// TwinCAT 3 PLC project Untitled1
// Title: EventBufferLibrary
// Company: Runtimevic SL
// Author: Víctor Durán Muñoz
// ProjectVersion: 1.0.0
// Description: victorduranm@hotmail.com
// ProgramVersion: 3.1.4023.0
// libraries:
//   Tc2_Standard, * (Beckhoff Automation GmbH)
//   Tc2_System, * (Beckhoff Automation GmbH)
//   Tc2_Utilities, * (Beckhoff Automation GmbH)
//   Tc3_EventLogger, * (Beckhoff Automation GmbH)
//   Tc3_Module, * (Beckhoff Automation GmbH)
//   TcUnit, * (www.tcunit.org)
// project tree:
//   / Demostration_1.TcTTO, PlcTask.TcTTO
//   DUTs/ E_EventType.TcDUT, ST_Event.TcDUT
//   POUs/ Demostration.TcPOU, EventLogger.TcPOU, FB_CsvPersistentEventStorage.TcPOU, FB_EventBuffer.TcPOU, FB_XmlPersistentEventStorage.TcPOU, I_PersistentEventStorage.TcIO, UpdateEventTimestampWithSystemTime.TcPOU
//   Project Information/ F_GetCompany.TcPOU, F_GetTitle.TcPOU, F_GetVersion.TcPOU
//   Test/ FB_EventBuffer_Test.TcPOU, PRG_TEST.TcPOU
//   Version/ Global_Version.TcGVL
// real-time tasks:
//   TASK PlcTask: cycle T#10ms, priority 20, ADS port 350
//   TASK Demostration: cycle T#10ms, priority 2, ADS port 352

CONFIGURATION Untitled1
    RESOURCE PLC ON TwinCAT3
        TASK Demostration_1(INTERVAL := T#10ms, PRIORITY := 2);
        TASK PlcTask(INTERVAL := T#10ms, PRIORITY := 20);
        PROGRAM Demostration WITH Demostration_1 : Demostration;
        PROGRAM PRG_TEST WITH PlcTask : PRG_TEST;
    END_RESOURCE
END_CONFIGURATION

// ---- DUTs/E_EventType.TcDUT
{attribute 'qualified_only'}
{attribute 'strict'}
TYPE E_EventType :
(
	Alarm :=0,
	Message :=1
);
END_TYPE

// ---- DUTs/ST_Event.TcDUT
TYPE ST_Event :
STRUCT
	eEventType :E_EventType;
	eEventSeverity: Tc3_EventLogger.TcEventSeverity;
	nEventIdentity: UDINT;
	sEventText: STRING(255);
	dtTimestamp: DATE_AND_TIME;
END_STRUCT
END_TYPE

// ---- Version/Global_Version.TcGVL
{attribute 'TcGenerated'}
{attribute 'no-analysis'}
{attribute 'linkalways'}
// This function has been automatically generated from the project information.
VAR_GLOBAL CONSTANT
	{attribute 'const_non_replaced'}
	stLibVersion_EventBufferLibrary : ST_LibVersion := (iMajor := 1, iMinor := 0, iBuild := 0, iRevision := 0, nFlags := 0, sVersion := '1.0.0');
END_VAR

// ---- POUs/I_PersistentEventStorage.TcIO
INTERFACE I_PersistentEventStorage

METHOD StoreEvent
VAR_INPUT
	stEvent : ST_Event;
END_VAR
END_METHOD

END_INTERFACE

// ---- POUs/Demostration.TcPOU
PROGRAM Demostration
VAR
	bBoolean : BOOL := FALSE;
	
	// Event #1
	eEventType1 :E_EventType := E_EventType.Alarm;
	eEventSeverity1: Tc3_EventLogger.TcEventSeverity := Tc3_EventLogger.TcEventSeverity.Error;
	nEventIdentity1: UDINT := 42;
	sEventText1: STRING(255) := 'this is a scary event #1';
	
	// Event #2
	eEventType2 :E_EventType := E_EventType.Alarm;
	eEventSeverity2: Tc3_EventLogger.TcEventSeverity := Tc3_EventLogger.TcEventSeverity.Error;
	nEventIdentity2: UDINT := 43;
	sEventText2: STRING(255) := 'this is a scary event #2';
	
	// Event #3
	eEventType3 :E_EventType := E_EventType.Alarm;
	eEventSeverity3: Tc3_EventLogger.TcEventSeverity := Tc3_EventLogger.TcEventSeverity.Error;
	nEventIdentity3: UDINT := 44;
	sEventText3: STRING(255) := 'this is a scary event #3';	
	
	
	BufferArray : ARRAY[0..(nMAXIMUM_NUMBER_OF_EVENTS * (SIZEOF(ST_Event) + nMEMORY_RING_BUFFER_INTERNAL_EXTRA_SPACING))] OF BYTE;
	fbEventBuffer : FB_EventBuffer(ADR(BufferArray),SIZEOF(BufferArray));	
	fbXmlPersistentEventStorage : FB_XmlPersistentEventStorage;	
	fbCsvPersistentEventStorage : FB_CsvPersistentEventStorage(fbEventBuffer);
//	EventLogger : EventLogger(fbXmlPersistentEventStorage);
	EventLogger : EventLogger(fbCsvPersistentEventStorage);
END_VAR
VAR CONSTANT
	nMAXIMUM_NUMBER_OF_EVENTS : UDINT := 10; 
	nMEMORY_RING_BUFFER_INTERNAL_EXTRA_SPACING : UDINT := 8;
END_VAR

IF bBoolean THEN
	EventLogger.AddEvent(eEventType1, eEventSeverity1, nEventIdentity1, sEventText1);
	EventLogger.AddEvent(eEventType2, eEventSeverity2, nEventIdentity2, sEventText2);
	EventLogger.AddEvent(eEventType3, eEventSeverity3, nEventIdentity3, sEventText3);
//	EventLogger.AddEvent(eEventType1, eEventSeverity1, nEventIdentity1, sEventText1);
	bBoolean := FALSE;
END_IF

fbCsvPersistentEventStorage();

END_PROGRAM

// ---- POUs/FB_EventBuffer.TcPOU
FUNCTION_BLOCK FB_EventBuffer
VAR
	fbMemRingBuffer			: Tc2_Utilities.FB_MemRingBuffer;
	pPointerToArrayBuffer 	: POINTER TO BYTE;
	nSizeOfArrayBuffer    	: UDINT;
END_VAR

METHOD PUBLIC AddEvent
VAR_INPUT
	stEvent : ST_Event;
END_VAR
VAR_OUTPUT
	bOk: BOOL; //
END_VAR
fbMemRingBuffer.A_AddTail(pWrite  := ADR(stEvent),
    					  cbWrite := SIZEOF(stEvent),  					
    					  pBuffer := pPointerToArrayBuffer,
    					  cbBuffer:= nSizeOfArrayBuffer);
						  
bOk:= fbMemRingBuffer.bOk;
END_METHOD

METHOD FB_init : BOOL
VAR_INPUT
	bInitRetains : BOOL; // if TRUE, the retain variables are initialized (warm start / cold start)
	bInCopyCode : BOOL;  // if TRUE, the instance afterwards gets moved into the copy code (online change)
	pPointerToArrayBuffer : POINTER TO BYTE;
	nSizeOfArrayBuffer    : UDINT;
END_VAR
THIS^.pPointerToArrayBuffer	:= pPointerToArrayBuffer;
THIS^.nSizeOfArrayBuffer    := nSizeOfArrayBuffer;
END_METHOD

METHOD PUBLIC GetAndRemoveEvent
VAR_OUTPUT
	stEvent : ST_Event;
	bOk  : BOOL;
END_VAR
fbMemRingBuffer.A_RemoveHead (pRead  := ADR(stEvent),
    					      cbRead := SIZEOF(stEvent),  					
    					      pBuffer := pPointerToArrayBuffer,
    					      cbBuffer:= nSizeOfArrayBuffer);
						  
bOk:= fbMemRingBuffer.bOk;
END_METHOD

METHOD PUBLIC GetNumberOfEvents : UDINT
GetNumberOfEvents := fbMemRingBuffer.nCount;
END_METHOD

END_FUNCTION_BLOCK

// ---- POUs/FB_XmlPersistentEventStorage.TcPOU
FUNCTION_BLOCK FB_XmlPersistentEventStorage IMPLEMENTS I_PersistentEventStorage
VAR_INPUT
END_VAR
VAR_OUTPUT
END_VAR
VAR
END_VAR

{warning 'add method implementation '}
METHOD StoreEvent
VAR_INPUT
	stEvent	: ST_Event;
END_VAR
// Here is there XML-Writing is supposed to be done
//Were is where the FB_XmlPersistentEventStorage se debe implementar el codigo aqui.
END_METHOD

END_FUNCTION_BLOCK

// ---- POUs/FB_CsvPersistentEventStorage.TcPOU
FUNCTION_BLOCK FB_CsvPersistentEventStorage IMPLEMENTS I_PersistentEventStorage
VAR
	fbFileOpen : FB_FileOpen := (sPathName := 'C:\Events.log', 
								 nMode := FOPEN_MODEAPPEND OR FOPEN_MODETEXT);
	fbFilePuts : FB_FilePuts;	
	fbFileClose : FB_FileClose;						 
	eWriteState : (WAIT_FOR_EVENT, FILE_OPEN_TRIGGER, FILE_OPEN, WRITE_EVENT_TRIGGER, WRITE_EVENT, FILE_CLOSE_TRIGGER, FILE_CLOSE, CLEAR_FILE_FB, ERROR);
	//stEventWrittenToFile : ST_Event;
	
	CsvString : T_MaxString;
	stEventFromBuffer : ST_Event;
	fbEventBuffer : REFERENCE TO FB_EventBuffer;
	bOkIgnore : BOOL;
END_VAR

CASE eWriteState OF
	WAIT_FOR_EVENT :
		//Do Anything
		IF fbEventBuffer.GetNumberOfEvents() > 0 THEN
			eWriteState := FILE_OPEN_TRIGGER;
		END_IF
		
	FILE_OPEN_TRIGGER :
		fbFileOpen(bExecute := TRUE);
		eWriteState := FILE_OPEN;
		
	FILE_OPEN :
		IF fbFileOpen.bError THEN
			eWriteState := ERROR;
		ELSIF NOT fbFileOpen.bBusy AND fbFileOpen.hFile <> 0 THEN
			eWriteState := WRITE_EVENT_TRIGGER;
		END_IF		
            fbFileOpen(bExecute := FALSE);	
		
	WRITE_EVENT_TRIGGER :
		eWriteState := FILE_OPEN_TRIGGER;
		fbEventBuffer.GetAndRemoveEvent(stEvent=> stEventFromBuffer, bOk=>bOkIgnore);
		CsvString := CreateCsvString(stEvent := stEventFromBuffer);
		fbFilePuts(bExecute := TRUE, 
				   sLine := CsvString,
				   hFile := fbFileOpen.hFile);
		eWriteState := WRITE_EVENT;
		
	WRITE_EVENT :
		IF fbFilePuts.bError THEN
			eWriteState := ERROR;
		ELSIF NOT fbFilePuts.bBusy THEN
			eWriteState := FILE_CLOSE_TRIGGER;
		END_IF			
		fbFilePuts(bExecute := FALSE);


	FILE_CLOSE_TRIGGER :
		fbFileClose(bExecute := TRUE,
					hFile := fbFileOpen.hFile);
		eWriteState := FILE_CLOSE;
		
	FILE_CLOSE :
	    IF fbFileClose.bError THEN
		    eWriteState := ERROR;
	    ELSIF NOT fbFileClose.bBusy THEN
		    eWriteState := WAIT_FOR_EVENT;
	    END_IF
	    fbFileClose(bExecute := FALSE);

	CLEAR_FILE_FB:
		fbFileOpen(bExecute := FALSE);
		fbFilePuts(bExecute := FALSE);
		fbFileClose(bExecute := FALSE);
		eWriteState := FILE_OPEN_TRIGGER;
		
	ERROR :
		//Do Nothing
END_CASE

METHOD PRIVATE CreateCsvString : T_MaxString
VAR_INPUT
	stEvent : REFERENCE TO ST_Event;
END_VAR
VAR
	TempString : T_MaxString;
//	count:  INT;
END_VAR
//TempString := TO_STRING(count +1);
//TempString := CONCAT(STR1:= TempString, STR2:= ',');
//TempString := CONCAT(STR1:= TempString, STR2:= TO_STRING(stEvent.eEventType));

TempString := TO_STRING(stEvent.eEventType);
TempString := CONCAT(STR1:= TempString, STR2:= ',');
TempString := CONCAT(STR1:= TempString, STR2:= TO_STRING(stEvent.eEventSeverity));
TempString := CONCAT(STR1:= TempString, STR2:= ',');
TempString := CONCAT(STR1:= TempString, STR2:= TO_STRING(stEvent.nEventIdentity));
TempString := CONCAT(STR1:= TempString, STR2:= ',');
TempString := CONCAT(STR1:= TempString, STR2:=  stevent.sEventText);
TempString := CONCAT(STR1:= TempString, STR2:= ',');
TempString := CONCAT(STR1:= TempString, STR2:=  TO_STRING(stEvent.dtTimestamp));
TempString := CONCAT(STR1:= TempString, STR2:=  '$N');

CreateCsvString := TempString;
END_METHOD

METHOD FB_init : BOOL
VAR_INPUT
	bInitRetains : BOOL; // if TRUE, the retain variables are initialized (warm start / cold start)
	bInCopyCode : BOOL;  // if TRUE, the instance afterwards gets moved into the copy code (online change)
	fbEventBuffer : REFERENCE TO FB_EventBuffer;
END_VAR
THIS^.fbEventBuffer REF= fbEventBuffer;
END_METHOD


METHOD StoreEvent
VAR_INPUT
	stEvent	: ST_Event;
END_VAR
VAR
	bOkIgnore : BOOL;
END_VAR
(*
IF eWriteState = WAIT_FOR_EVENT THEN
	eWriteState := FILE_OPEN_TRIGGER;
	stEventWrittenToFile := stEvent;
END_IF
*)
fbEventBuffer.AddEvent(stEvent:= stEvent, bOk=>bOkIgnore);
END_METHOD

END_FUNCTION_BLOCK

// ---- POUs/EventLogger.TcPOU
FUNCTION_BLOCK EventLogger
VAR
	EventBuffer : ARRAY[1..MAXIMUM_SIZE_OF_EVENT_BUFFER] OF ST_Event;
	CurrentEventBufferIndex : INT :=0;
	
	_PersistentEventStorage : I_PersistentEventStorage;
END_VAR
VAR CONSTANT
	MAXIMUM_SIZE_OF_EVENT_BUFFER : INT := 100;
END_VAR

(* Returns TRUE if add was succesful and FALSE if buffer is full *)
METHOD PUBLIC AddEvent : BOOL
VAR_INPUT
	eEventType :E_EventType;
	eEventSeverity: Tc3_EventLogger.TcEventSeverity;
	nEventIdentity: UDINT;
	sEventText: STRING(255);
END_VAR
IF NOT IsEventBufferFull() THEN
	CurrentEventBufferIndex := CurrentEventBufferIndex + 1;
	EventBuffer[CurrentEventBufferIndex].eEventType := eEventType;
	EventBuffer[CurrentEventBufferIndex].eEventSeverity := eEventSeverity;
	EventBuffer[CurrentEventBufferIndex].nEventIdentity := nEventIdentity;
	EventBuffer[CurrentEventBufferIndex].sEventText := sEventText;
	UpdateEventTimestampWithSystemTime(stEvent := EventBuffer[CurrentEventBufferIndex]);	
//	AddEvent := TRUE;
//ELSE
//	AddEvent := FALSE;
END_IF

AddEvent := NOT IsEventBufferFull();

//Here we want to store the event persistently
_PersistentEventStorage.StoreEvent(EventBuffer[CurrentEventBufferIndex]);
END_METHOD

METHOD FB_init : BOOL
VAR_INPUT
	bInitRetains : BOOL; // if TRUE, the retain variables are initialized (warm start / cold start)
	bInCopyCode : BOOL;  // if TRUE, the instance afterwards gets moved into the copy code (online change)
	iPersistentEventStorage :I_PersistentEventStorage;
END_VAR
_PersistentEventStorage := iPersistentEventStorage;
END_METHOD

METHOD PRIVATE IsEventBufferFull : BOOL
IsEventBufferFull := (CurrentEventBufferIndex + 1) > MAXIMUM_SIZE_OF_EVENT_BUFFER;
END_METHOD

END_FUNCTION_BLOCK

// ---- POUs/UpdateEventTimestampWithSystemTime.TcPOU
FUNCTION UpdateEventTimestampWithSystemTime
VAR_INPUT
	stEvent : REFERENCE TO ST_Event;
END_VAR
VAR
	fbGETSYSTEMTIME : GETSYSTEMTIME;
	stFileTime		: T_FILETIME;
END_VAR

fbGETSYSTEMTIME(timeLoDW=> stFileTime.dwLowDateTime , timeHiDW=> stFileTime.dwHighDateTime);

stEvent.dtTimestamp:= FILETIME_TO_DT(fileTime := stFileTime);

END_FUNCTION

// ---- Test/PRG_TEST.TcPOU
PROGRAM PRG_TEST
VAR
	fbEventBuffer_Test : FB_EventBuffer_Test;
END_VAR

TcUnit.RUN();

END_PROGRAM

// ---- Test/FB_EventBuffer_Test.TcPOU
FUNCTION_BLOCK FB_EventBuffer_Test EXTENDS TcUnit.FB_TestSuite
VAR
END_VAR

AddThreeEventsExceptAllToBeCorrectAndSuccessfull();
AddFourEventsExpectAllToBeAddedExceptTheLastOne();
AddOneEventGetTwoExpectTheSecondOneToFail();

METHOD PRIVATE AddFourEventsExpectAllToBeAddedExceptTheLastOne
VAR
	ArrayBuffer : ARRAY[0..(3 * (SIZEOF(ST_Event) + 8))] OF BYTE;
	EventBuffer : FB_EventBuffer(pPointerToArrayBuffer:= ADR(ArrayBuffer), nSizeOfArrayBuffer:= SIZEOF(ArrayBuffer));
	
	// Event #1
	stEvent1: ST_Event :=	(eEventType := E_EventType.Alarm,
							eEventSeverity:= Tc3_EventLogger.TcEventSeverity.Critical,
							nEventIdentity:= 42,
							sEventText:= 'Hi there!',
							dtTimestamp:= DT#2016-01-07-06:28:11);	
							
	bOk 			: BOOL;								
END_VAR
TEST('AddFourEventsExpectAllToBeAddedExceptTheLastOne');

// Event #1
EventBuffer.AddEvent(stEvent:= stEvent1, bOk=> bOk);
AssertTrue(Condition:=bOk, Message:= 'Should have been added successfully #1');

// Event #2
EventBuffer.AddEvent(stEvent:= stEvent1, bOk=> bOk);
AssertTrue(Condition:=bOk, Message:= 'Should have been added successfully #2');

// Event #3
EventBuffer.AddEvent(stEvent:= stEvent1, bOk=> bOk);
AssertTrue(Condition:=bOk, Message:= 'Should have been added successfully #3');

// Event #4
EventBuffer.AddEvent(stEvent:= stEvent1, bOk=> bOk);
AssertFalse(Condition:=bOk, Message:= 'Should NOT have been added successfully');


TEST_FINISHED();
END_METHOD

METHOD PRIVATE AddOneEventGetTwoExpectTheSecondOneToFail
VAR
	ArrayBuffer : ARRAY[0..(3 * (SIZEOF(ST_Event) + 8))] OF BYTE;
	EventBuffer : FB_EventBuffer(pPointerToArrayBuffer:= ADR(ArrayBuffer), nSizeOfArrayBuffer:= SIZEOF(ArrayBuffer));
	
	// Event #1
	stEvent1: ST_Event :=	(eEventType := E_EventType.Alarm,
							eEventSeverity:= Tc3_EventLogger.TcEventSeverity.Critical,
							nEventIdentity:= 42,
							sEventText:= 'Hi there!',
							dtTimestamp:= DT#2016-01-07-06:28:11);	
							
	bOkReturn 			: BOOL;	
	stEventReturn		: ST_Event;		
END_VAR
TEST('AddOneEventGetTwoExpectTheSecondOneToFail');

// Round #1
EventBuffer.AddEvent(stEvent:= stEvent1, bOk=> bOkReturn);
EventBuffer.GetAndRemoveEvent(stEvent=> stEventReturn, bOk=>bOkReturn);
AssertTrue(Condition:=bOkReturn, Message:= 'Expected OK to be true');

// Round #2
EventBuffer.GetAndRemoveEvent(stEvent=> stEventReturn, bOk=>bOkReturn);
AssertFalse(Condition:=bOkReturn, Message:= 'Expected OK to be false');

TEST_FINISHED();
END_METHOD

METHOD PRIVATE AddThreeEventsExceptAllToBeCorrectAndSuccessfull
VAR
	ArrayBuffer : ARRAY[0..(3 * (SIZEOF(ST_Event) + 8))] OF BYTE;
	EventBuffer : FB_EventBuffer(pPointerToArrayBuffer:= ADR(ArrayBuffer), nSizeOfArrayBuffer:= SIZEOF(ArrayBuffer));
	
	// Event #1
	stEvent1: ST_Event :=	(eEventType := E_EventType.Alarm,
							eEventSeverity:= Tc3_EventLogger.TcEventSeverity.Critical,
							nEventIdentity:= 42,
							sEventText:= 'Hi there!',
							dtTimestamp:= DT#2016-01-07-06:28:11);
							
	// Event #2
	stEvent2: ST_Event :=	(eEventType := E_EventType.Message,
							eEventSeverity:= Tc3_EventLogger.TcEventSeverity.Info,
							nEventIdentity:= 43,
							sEventText:= 'Hi there2',
							dtTimestamp:= DT#2016-02-07-06:28:12);

	// Event #3
	stEvent3: ST_Event :=	(eEventType := E_EventType.Alarm,
							eEventSeverity:= Tc3_EventLogger.TcEventSeverity.Error,
							nEventIdentity:= 44,
							sEventText:= 'Hi there3',
							dtTimestamp:= DT#2016-03-07-06:28:13);	

	bOk 			: BOOL;	
	nNumberOfEvents	: UDINT;		
	stEvent 		: ST_Event;			
END_VAR
TEST('AddThreeEventsExceptAllToBeCorrectAndSuccessfull');

//Add Event #1
EventBuffer.AddEvent(stEvent:= stEvent1, bOk=> bOk);
AssertTrue(Condition:=bOk, Message:= 'Add event #1 was not OK');
nNumberOfEvents := EventBuffer.GetNumberOfEvents();
AssertEquals_UDINT(Expected:= 1, Actual:= nNumberOfEvents, Message:='Expected one event');

//Add Event #2
EventBuffer.AddEvent(stEvent:= stEvent2, bOk=> bOk);
AssertTrue(Condition:=bOk, Message:= 'Add event #2 was not OK');
nNumberOfEvents := EventBuffer.GetNumberOfEvents();
AssertEquals_UDINT(Expected:= 2, Actual:= nNumberOfEvents, Message:='Expected two events');

//Add Event #3
EventBuffer.AddEvent(stEvent:= stEvent3, bOk=> bOk);
AssertTrue(Condition:=bOk, Message:= 'Add event #3 was not OK');
nNumberOfEvents := EventBuffer.GetNumberOfEvents();
AssertEquals_UDINT(Expected:= 3, Actual:= nNumberOfEvents, Message:='Expected three events');

// Read Event #1
EventBuffer.GetAndRemoveEvent(stEvent=> stEvent, bOk=>bOk);
AssertTrue(Condition:=bOk, Message:= 'Read of event #1 was not successful');
AssertEquals_UDINT(Expected:= 2, Actual:= EventBuffer.GetNumberOfEvents(), Message:='Expected two events');
AssertEquals_INT(Expected:= E_EventType.Alarm, Actual:= stEvent.eEventType, Message:='Expected event type Alarm');
AssertEquals_INT(Expected:= TcEventSeverity.Critical, Actual:= stEvent.eEventSeverity, Message:='Expected event severity Critical');
AssertEquals_UDINT(Expected:= 42, Actual:= stEvent.nEventIdentity, Message:='Expected event identity 42');
AssertEquals_STRING(Expected:= 'Hi there!', Actual:= stEvent.sEventText, Message:='Expected: Hi there!');
AssertEquals_DATE_AND_TIME(Expected:= stEvent1.dtTimestamp, Actual:= stEvent.dtTimestamp, Message:='Expected: DT#2016-01-07-06:28:11');

// Read Event #2
EventBuffer.GetAndRemoveEvent(stEvent=> stEvent, bOk=>bOk);
AssertTrue(Condition:=bOk, Message:= 'Read of event #2 was not successful');
AssertEquals_UDINT(Expected:= 1, Actual:= EventBuffer.GetNumberOfEvents(), Message:='Expected one events');
AssertEquals_INT(Expected:= E_EventType.Message, Actual:= stEvent.eEventType, Message:='Expected event type Message');
AssertEquals_INT(Expected:= TcEventSeverity.info, Actual:= stEvent.eEventSeverity, Message:='Expected event severity Info');
AssertEquals_UDINT(Expected:= stEvent2.nEventIdentity, Actual:= stEvent.nEventIdentity, Message:='Expected event identity 43');
AssertEquals_STRING(Expected:= 'Hi there2', Actual:= stEvent.sEventText, Message:='Expected: Hi there2');
AssertEquals_DATE_AND_TIME(Expected:= stEvent2.dtTimestamp, Actual:= stEvent.dtTimestamp, Message:='Expected: DT#2016-02-07-06:28:12');

// Read Event #3
EventBuffer.GetAndRemoveEvent(stEvent=> stEvent, bOk=>bOk);
AssertTrue(Condition:=bOk, Message:= 'Read of event #3 was not successful');
AssertEquals_UDINT(Expected:= 0, Actual:= EventBuffer.GetNumberOfEvents(), Message:='Expected cero events');
AssertEquals_INT(Expected:= E_EventType.Alarm, Actual:= stEvent.eEventType, Message:='Expected event type Alarm');
AssertEquals_INT(Expected:= TcEventSeverity.Error, Actual:= stEvent.eEventSeverity, Message:='Expected event severity Error');
AssertEquals_UDINT(Expected:= stEvent3.nEventIdentity, Actual:= stEvent.nEventIdentity, Message:='Expected event identity 44');
AssertEquals_STRING(Expected:= stEvent3.sEventText, Actual:= stEvent.sEventText, Message:='Expected: Hi there3');
AssertEquals_DATE_AND_TIME(Expected:= stEvent3.dtTimestamp, Actual:= stEvent.dtTimestamp, Message:='Expected: DT#2016-03-07-06:28:13');

TEST_FINISHED();
END_METHOD

END_FUNCTION_BLOCK

// ---- Project Information/F_GetCompany.TcPOU
// This function has been automatically generated from the project information.
{attribute 'signature_flag' := '1073741824'}
{attribute 'TcGenerated'}
{attribute 'no-analysis'}
FUNCTION F_GetCompany : WSTRING
VAR_INPUT
	
END_VAR

F_GetCompany := "Runtimevic SL";

END_FUNCTION

// ---- Project Information/F_GetTitle.TcPOU
// This function has been automatically generated from the project information.
{attribute 'signature_flag' := '1073741824'}
{attribute 'TcGenerated'}
{attribute 'no-analysis'}
FUNCTION F_GetTitle : WSTRING
VAR_INPUT
	
END_VAR

F_GetTitle := "EventBufferLibrary";

END_FUNCTION

// ---- Project Information/F_GetVersion.TcPOU
// This function has been automatically generated from the project information.
{attribute 'signature_flag' := '1073741824'}
{attribute 'TcGenerated'}
{attribute 'no-analysis'}
FUNCTION F_GetVersion : ST_LibVersion
VAR_INPUT
	
END_VAR

F_GetVersion.iMajor := 1;
F_GetVersion.iMinor := 0;
F_GetVersion.iBuild := 0;
F_GetVersion.iRevision := 0;
F_GetVersion.sVersion := '1.0.0';
F_GetVersion.nFlags := 0;

END_FUNCTION
